// TIA Portal V16 export
// export: Created 2021-05-11T05:22:24.8939056Z, ExportSetting WithDefaults, DisplayName Totally Integrated Automation Portal, DisplayVersion V16, DisplayName TIA Portal Version Control Interface, DisplayVersion V16, DisplayName TIA Portal Openness, DisplayVersion V16, DisplayName STEP 7 Professional, DisplayVersion V16, DisplayName STEP 7 Safety, DisplayVersion V16, DisplayName WinCC Unified SCADA Engineering System, DisplayVersion V16
TYPE "PCT_TSA"
// stored: IsFailsafeCompliant false
   STRUCT
      AlarmeTempTransfoAuxSeuil1 : Bool;   // PCT-TK:
      AlarmeTempTransfoAuxSeuil2 : Bool;   // PCT-TK:
      SynthDefRelaisSondeProtectTSA : Bool;   // PCT-TK:
      Valeur_INT : Int;   // PCT-TK:
      Valeur_DINT : DInt;   // PCT-TK:
      Valeur_Flottant : Real;   // PCT-TK:
   END_STRUCT;
END_TYPE
